FUNCTION_BLOCK Starting_State  IMPLEMENTS ITF_State
VAR_INPUT
END_VAR
VAR_OUTPUT
END_VAR
VAR
	pPML_Base : POINTER TO PML_StatePattern_Base;
	_stateMachine : IPmlStateMachine;
END_VAR

METHOD Cycle : BOOL
VAR_INPUT
END_VAR
_stateMachine.SetStateComplete();
pPML_Base^.SetState(pPML_Base^.execute);
END_METHOD

METHOD FB_init : BOOL
VAR_INPUT
	bInitRetains : BOOL; // if TRUE, the retain variables are initialized (warm start / cold start)
	bInCopyCode : BOOL;  // if TRUE, the instance afterwards gets moved into the copy code (online change)
	pPML_Base : POINTER TO PML_StatePattern_Base;
	statemachine : IPmlStateMachine;
END_VAR
_stateMachine := statemachine;
THIS^.pPML_Base := pPML_Base;
END_METHOD

END_FUNCTION_BLOCK

(* stored: Version 1.1.0.1, ProductVersion 3.1.4024.11
   POU Starting_State: Id {90b2215b-0be1-470f-a673-dc26b3c8a557}, SpecialFunc None
   Method Cycle: Id {eea347af-0d21-4663-a3a3-eccec491c26b}
   Method FB_init: Id {0ef899d2-aa77-4bb8-b467-3190895e6d8a} *)
